// Block: A0301_Trasporto_PERS

DATA_BLOCK A0301_Trasporto_PERS
VERSION : 0.1
   NON_RETAIN
   VAR
      Par : Struct
         Ax : SpeedMachine_Par;
         Ax_Aut : A0301_Mach_Speed_Par;
      END_STRUCT;
   END_VAR

BEGIN
   // No initialization required
END_DATA_BLOCK
